PROGRAM MAIN
VAR
fbReadCoe : FB_Read70x1CoeData;
END_VAR

fbReadCoe(userNetId:= '172.21.148.67.2.1');

END_PROGRAM

(* stored: Version 1.1.0.1, ProductVersion 3.1.4022.18
   POU MAIN: Id {5c316f37-c00a-4846-b3a7-5df370ce17b6}, SpecialFunc None *)
